TYPE ST_SensirionFMStatus :
STRUCT
	

	iFlowTicks	:	INT;
	uiSensorOutput	: UINT;
	iState	:	INT;
	rFlow	:	REAL; // units of uL/min
	xOoR	:	BOOL; // Out of range
	xFMMode :	BOOL; // calib mode 0 = prec, 1 = extended
	xFlowValid	:	BOOL; // driver completes successfully
	abReply	:	ARRAY[1..500] OF BYTE;
	bAdr	:	BYTE; //Device address
	bStatus	:	BYTE; //Sensor status
(* Bit 0: 0: Sensor idle
		1: Sensor Busy
Bit 1: 	0: Continuous Measurement disabled
		1: Continuous Measurement enabled
Bit 2: (for Firmware . 1.3)
		0: Auto detection Measurement disabled
		1: Auto detection Measurement enabled
Bit 3: (for Firmware . 1.3)
		0: No Auto Measurement since last read out Status
		1: Auto Measurement finished since last read out Status, is set back to 0 after read out *)

END_STRUCT
END_TYPE

(* stored: Version 1.1.0.1, ProductVersion 3.1.0.26
   DUT ST_SensirionFMStatus: Id {167d0110-ce48-475a-b7ba-7b29f3e90a1e} *)
